FUNCTION_BLOCK FB_GetFifo
VAR_INPUT
END_VAR
VAR_OUTPUT
	bFIFO_Empty:BOOL;
	out_STRING:STRING(255);
END_VAR
VAR_IN_OUT
	DB:ST_String_FIFO;
END_VAR
VAR
END_VAR

bFIFO_Empty := FALSE;
IF DB.Count > 0 THEN
	out_STRING := DB.DB[DB.Output_Pointer];
	DB.DB[DB.Output_Pointer] := '';
	DB.Count := DB.Count - 1;

	DB.Output_Pointer := DB.Output_Pointer + 1;
	IF DB.Output_Pointer > DB.DataTop THEN
		DB.Output_Pointer := 0;
	END_IF

ELSE
	bFIFO_Empty := TRUE;
END_IF

END_FUNCTION_BLOCK

(* stored: Version 1.1.0.1, ProductVersion 3.1.4024.5
   POU FB_GetFifo: Id {856a7513-08fe-438f-b923-79134b901d3a}, SpecialFunc None *)
